# B&R Automation Studio project Palnik
Automation Studio 3.0.90.32 SP14

## Configuration 4PP481

### Task classes (Cpu.sw)
```
Cyclic#4:
  Palnik <- Palnik.prg
Libraries: standard
```

### IoMap.iom - PLC1/IoMap.iom
```iecst
(********************************************************************
 * COPYRIGHT --
 ********************************************************************
 * File: IoMap.iom
 * Author: User
 * Created: November 09, 2017
 ********************************************************************
 * IO mapping file
 ********************************************************************)
VAR_CONFIG
	Palnik.System.diStart AT %IX.SL1.SS1.IF1.ST2.DigitalInput01;
	Palnik.System.diStop AT %IX.SL1.SS1.IF1.ST2.DigitalInput02;
	Palnik.System.diEStop AT %IX.SL1.SS1.IF1.ST2.DigitalInput03;
	Palnik.Palnik[0].diFanStarter AT %IX.SL1.SS1.IF1.ST2.DigitalInput04;
	Palnik.Palnik[0].diAirFlow AT %IX.SL1.SS1.IF1.ST2.DigitalInput05;
	Palnik.Palnik[0].diFlameDetector AT %IX.SL1.SS1.IF1.ST2.DigitalInput06;
	Palnik.System.doSystemAktywny AT %QX.SL1.SS1.IF1.ST3.DigitalOutput01;
	Palnik.Palnik[0].doAirFan AT %QX.SL1.SS1.IF1.ST3.DigitalOutput02;
	Palnik.Palnik[0].doPilotValve AT %QX.SL1.SS1.IF1.ST3.DigitalOutput03;
	Palnik.Palnik[0].doMainValve AT %QX.SL1.SS1.IF1.ST3.DigitalOutput04;
	Palnik.Palnik[0].doIgniter AT %QX.SL1.SS1.IF1.ST3.DigitalOutput05;
END_VAR
```

## Configuration Simulation

### Task classes (Cpu.sw)
```
Cyclic#4:
  Palnik <- Palnik.prg
Libraries: AsIecCon, astime, standard
```

## Logical view

Binary libraries used (declarations not repeated): RUNTIME, Operator, AsIecCon, astime, standard

### Package Logical/Libraries - Global libraries

- Visualisation Logical/Visu (not shown)

### Program Logical/Palnik (IEC) - A new program

#### Palnik.ab - Implementation code
```automation-basic
(********************************************************************
 * COPYRIGHT -- Microsoft
 ********************************************************************
 * Program: Palnik
 * File: Palnik.ab
 * Author: Liss_1
 * Created: January 04, 2018
 ********************************************************************
 * Implementation of program Palnik
 ********************************************************************)

PROGRAM _INIT

END_PROGRAM

PROGRAM _CYCLIC

	//czujnik air flow - nie ma go na tym schemacie, ale jest gdzieś tam w zgięciu gdzie płynie air
	// normalnie jest otwarty

	//state init jest bezwarunkowy
	System.doSystemAktywny = ((System.diStart OR System.doSystemAktywny) AND NOT(System.diStop)) //dodac obsluge diEStop chyba
	SELECT
		STATE INIT // Oczekiwanie na akcje uzytkownika
			// operacje do wykonania
			//
			WHEN System.doSystemAktywny = TRUE
				NEXT AIRFAN

		STATE AIRFAN
			Palnik[0].doAirFan = TRUE

			Wait[1].IN = Palnik[0].diAirFlow
			Wait[1].ET = T#0s
			Wait[1].PT = T#3s
			Wait[1] FUB TON()
			WHEN (Palnik[0].diFanStarter = TRUE) AND (Wait[1].Q = TRUE)
				NEXT AIRING

		STATE AIRING
			Wait[0].IN = FALSE
			Wait[0].IN = TRUE
			Wait[0].ET = T#0s
			Wait[0].PT = T#10s
			Wait[0] FUB TON()
			WHEN Wait[0].Q = TRUE
				NEXT INITBURN

		STATE INITBURN

			i = i + 1
			WHEN i=5
				NEXT STOP

			WHEN TRUE
				NEXT IGNITION

		STATE IGNITION
			Wait[2].IN = FALSE
			Wait[2].IN = TRUE
			Wait[2].ET = T#0s
			Wait[2].PT = T#2s

			Palnik[0].doPilotValve = TRUE
			Palnik[0].doIgniter = TRUE
			Wait[2] FUB TON()
			WHEN (Wait[2].Q = TRUE)
				NEXT IGNITION2

		STATE IGNITION2
			Palnik[0].doIgniter = FALSE
			IF (Palnik[0].diFlameDetector = TRUE) THEN
				Palnik[0].doIgniter = FALSE
				Palnik[0].doMainValve = TRUE
				Palnik[0].doPilotValve = FALSE
				flag = TRUE
			ELSE
				Palnik[0].doIgniter = FALSE
				Palnik[0].doMainValve = FALSE
				Palnik[0].doPilotValve = FALSE
			ENDIF

			WHEN flag = TRUE
				NEXT BURN
			WHEN flag = FALSE
				NEXT BREAK

		STATE BREAK
			Wait[3].IN = FALSE
			Wait[3].IN = TRUE
			Wait[3].ET = T#0s
			Wait[3].PT = T#3s
			Wait[3] FUB TON()
			WHEN Wait[3].Q = TRUE
				NEXT INITBURN

		STATE BURN
			f1 = System.diStop
			f2 = System.diEStop
			f3 = Palnik[0].diAirFlow
			f4 = Palnik[0].diFlameDetector
			WHEN ((f1 = TRUE) OR (f2 = TRUE) OR (f3 = FALSE) OR (f4 = FALSE))
				NEXT STOP

		STATE STOP // wylaczenie wszystkiego
			Palnik[0].doMainValve = FALSE
			Palnik[0].doPilotValve = FALSE
			System.diStop = FALSE
			System.diEStop = FALSE
			System.diStart = FALSE
			i = 0
			Wait[0].IN = FALSE
			Wait[1].IN = FALSE
			Wait[2].IN = FALSE
			Wait[3].IN = FALSE
			Wait[4].IN = FALSE

			Wait[4].IN = TRUE
			Wait[4].ET = T#0s
			Wait[4].PT = T#10s
			Wait[4] FUB TON()

			WHEN (Wait[4].Q = TRUE)
				 NEXT STOPFINAL

		STATE STOPFINAL
			Palnik[0].doAirFan = FALSE
			IF ((Palnik[0].diFlameDetector = FALSE) AND (Palnik[0].doAirFan = FALSE)) THEN
				System.doSystemAktywny = FALSE
			ENDIF
			WHEN (System.doSystemAktywny = FALSE)
				NEXT INIT

	ENDSELECT

END_PROGRAM
```

#### Palnik.typ - Local data types
```iecst
(********************************************************************
 * COPYRIGHT -- Microsoft
 ********************************************************************
 * Program: Palnik
 * File: Palnik.typ
 * Author: Liss_1
 * Created: January 04, 2018
 ********************************************************************
 * Local data types of program Palnik
 ********************************************************************)

TYPE
	SystemStruct : 	STRUCT
		diStop : BOOL;
		diStart : BOOL;
		diEStop : BOOL;
		doSystemAktywny : BOOL;
	END_STRUCT;
	BurnerStruct : 	STRUCT
		diFanStarter : BOOL;
		doAirFan : BOOL;
		diAirFlow : BOOL;
		diFlameDetector : BOOL;
		doPilotValve : BOOL;
		doMainValve : BOOL;
		doIgniter : BOOL;
	END_STRUCT;
END_TYPE
```

#### Palnik.var - Local variables
```iecst
(********************************************************************
 * COPYRIGHT -- Microsoft
 ********************************************************************
 * Program: Palnik
 * File: Palnik.var
 * Author: Liss_1
 * Created: January 04, 2018
 ********************************************************************
 * Local variables of program Palnik
 ********************************************************************)
VAR
	Wait : ARRAY[0..10] OF TON := [11(0)];
	Palnik : ARRAY[0..10] OF BurnerStruct := [11(0)];
	System : SystemStruct := (0);
	i : INT := 0;
	flag : BOOL := FALSE;
	f4 : BOOL := FALSE;
	f3 : BOOL := FALSE;
	f2 : BOOL := FALSE;
	f1 : BOOL := FALSE;
END_VAR
```

Listed in the project but not available here: Logical/Global.typ, Logical/Global.var
